// TIA Portal V17 export
// export: Created 2022-07-20T07:01:27.2543437Z, ExportSetting WithDefaults, DisplayName Totally Integrated Automation Portal, DisplayVersion V17, DisplayName TIA Portal Openness, DisplayVersion V17, DisplayName TIA Portal Version Control Interface, DisplayVersion V17, DisplayName SINAMICS Startdrive Advanced, DisplayVersion V17, DisplayName SINAMICS Startdrive G130, G150, S120, S150, SINAMICS MV, S210, DisplayVersion V17, DisplayName SINAMICS Startdrive G110M, G120, G120C, G120D, G120P, G115D, DisplayVersion V17, DisplayName STEP 7 Professional, DisplayVersion V17, DisplayName STEP 7 Safety, DisplayVersion V17, DisplayName WinCC Advanced, DisplayVersion V17
FUNCTION_BLOCK "FB10270_HiwinDoorActuatorManager"   // FB10270, LAD
{ S7_Optimized_Access := 'TRUE' }
VERSION : 0.1
// stored: AutoNumber false, IsIECCheckEnabled false, IsRetainMemResEnabled false, MemoryReserve 100, SetENOAutomatically false, UDAEnableTagReadback false
   VAR_INPUT
      RequestButtonDoorActivation { ExternalAccessible := 'False'; ExternalVisible := 'False'; ExternalWritable := 'False'} : Bool;
      AuthorizeToOpenDoor : Bool;
      ClosedPositionLimitSwitch : Bool;
   END_VAR
   VAR_OUTPUT
      ActuatorGoToOpenPosition : Bool;
      ActuatorGoToClosePosition { ExternalAccessible := 'False'; ExternalVisible := 'False'; ExternalWritable := 'False'} : Bool;
      ButtonLight : Bool;
      IsInClosedPosition : Bool;
      IsInOpenedPosition : Bool;
      ActuatorInError : Bool;
   END_VAR
   VAR
      ShortPushDetected : Bool;
      LongPushDetected : Bool;
      DoorActuatorManagementStateDiagram : Int;
      R_TRIG_ShortPushDetected : R_TRIG;
      R_TRIG_LongPushDetected { S7_SetPoint := 'True'} : R_TRIG;
      TON_GoToOpenPositionTime { S7_SetPoint := 'True'} : TON_TIME;
      FB10001_PulseControl_Instance { S7_SetPoint := 'True'} : "FB10001_PulseControl";
      FB10041_DetectKindOfPush_Instance { S7_SetPoint := 'True'} : "FB10041_DetectKindOfPush";
   END_VAR
   VAR CONSTANT
      WAIT_FOR_ACTUATOR_COMMAND : Int := 0;
      ACTUATOR_GO_TO_OPEN_POSITION : Int := 10;
      ACTUATOR_GO_TO_CLOSE_POSITION : Int := 20;
      ACTUATOR_COMMAND_DONE : Int := 30;
   END_VAR
BEGIN

REGION Network 1 (SCL): FirstScan
   IF "FirstScan"THEN
       ;
   END_IF;
END_REGION

REGION Network 2 (SCL): Edge Signals & Timers
   REGION EDGE SIGNALS
       #R_TRIG_ShortPushDetected(CLK := #ShortPushDetected AND #AuthorizeToOpenDoor);
       #R_TRIG_LongPushDetected(CLK := #LongPushDetected AND #RequestButtonDoorActivation);
   END_REGION

   REGION TIMERS
       #TON_GoToOpenPositionTime(IN := #ActuatorGoToOpenPosition,
                                 PT := T#25s);
   END_REGION
END_REGION

REGION Network 3: Kind Of Push Button Management
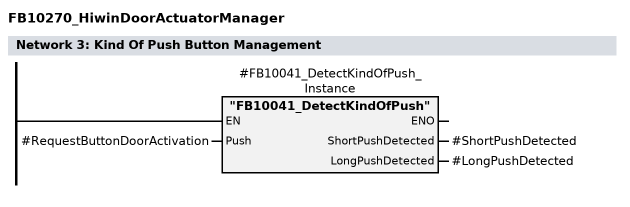
   RUNG wire#powerrail
      #FB10041_DetectKindOfPush_Instance(Push := #RequestButtonDoorActivation, ShortPushDetected => #ShortPushDetected, LongPushDetected => #LongPushDetected)
   END_RUNG
   // the same network as SCL:
   #FB10041_DetectKindOfPush_Instance(Push := #RequestButtonDoorActivation,   // "FB10041_DetectKindOfPush"
                           ShortPushDetected => #ShortPushDetected,
                           LongPushDetected => #LongPushDetected);
END_REGION

REGION Network 4 (SCL): Button Led Management
   IF #AuthorizeToOpenDoor THEN
       #ButtonLight := TRUE;
   ELSIF NOT (#AuthorizeToOpenDoor) AND #ClosedPositionLimitSwitch THEN
       #FB10001_PulseControl_Instance(Time_On := T#300ms,
                                      Time_Off := T#300ms,
                                      Signal := #DoorActuatorManagementStateDiagram = #ACTUATOR_GO_TO_OPEN_POSITION OR
                                      #DoorActuatorManagementStateDiagram = #ACTUATOR_GO_TO_CLOSE_POSITION,
                                      SignalPulsed => #ButtonLight);
   ELSE
       #ButtonLight := FALSE;
   END_IF;
END_REGION

REGION Network 5 (SCL): Actuator Management
   CASE #DoorActuatorManagementStateDiagram OF
       #WAIT_FOR_ACTUATOR_COMMAND:
           IF #R_TRIG_ShortPushDetected.Q THEN
               #DoorActuatorManagementStateDiagram := #ACTUATOR_GO_TO_OPEN_POSITION;
           ELSIF #R_TRIG_LongPushDetected.Q THEN
               #DoorActuatorManagementStateDiagram := #ACTUATOR_GO_TO_CLOSE_POSITION;
           END_IF;
       #ACTUATOR_GO_TO_OPEN_POSITION:
           #ActuatorGoToClosePosition := FALSE;
           #ActuatorGoToOpenPosition := NOT (#ActuatorGoToOpenPosition);
           #DoorActuatorManagementStateDiagram := #ACTUATOR_COMMAND_DONE;
       #ACTUATOR_GO_TO_CLOSE_POSITION:
           IF #RequestButtonDoorActivation THEN
               #ActuatorGoToOpenPosition := FALSE;
               #ActuatorGoToClosePosition := TRUE;
           ELSIF NOT (#RequestButtonDoorActivation) OR NOT (#ClosedPositionLimitSwitch) THEN
               #ActuatorGoToOpenPosition := FALSE;
               #ActuatorGoToClosePosition := FALSE;
               #DoorActuatorManagementStateDiagram := #ACTUATOR_COMMAND_DONE;
           END_IF;
       #ACTUATOR_COMMAND_DONE:
           #DoorActuatorManagementStateDiagram := #WAIT_FOR_ACTUATOR_COMMAND;
   END_CASE;
END_REGION

REGION Network 6 (SCL): Actuator Safety Management
   IF #TON_GoToOpenPositionTime.Q THEN
       #ActuatorGoToOpenPosition := FALSE;
   END_IF;
END_REGION

REGION Network 7 (SCL): Actuator States Management
   #IsInClosedPosition := #ClosedPositionLimitSwitch;
   #IsInOpenedPosition := NOT (#ClosedPositionLimitSwitch);
END_REGION
END_FUNCTION_BLOCK
